Universal Robots PolyScope program: pos5.urp

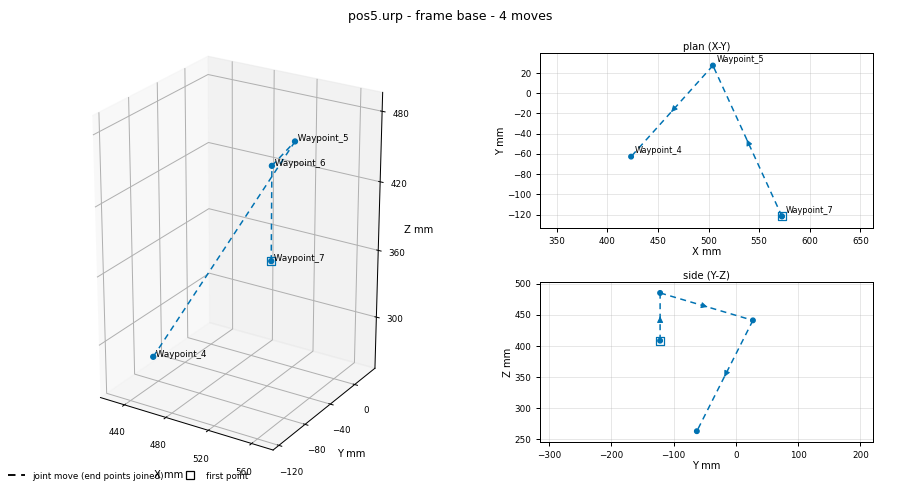
[picture p0: tool path of pos5.urp in frame base, 4 of 4 moves have a stored position in this frame; points joined in program order, loops and branches not executed]
Program pos5 (installation=default directory=/programs/Nicolas_Arteaga/quality createdIn=5.12.4.1101661 lastSavedIn=5.12.4.1101661 robotSerialNumber=20225502378)
Calibrated DH parameters: a=[0.00022, -0.425328, -0.389701, 0.000059, 0.000065, 0]; d=[0.162608, 0.803456, 9.992211, -10.662202, 0.099702, 0.099559]; alpha=[1.570756, 0.001543, 0.004316, 1.570651, -1.570122, 0]; deltaTheta=[0, 0.002917, 0.116094, -0.119008, 0, -0.000001]
Robot Program (runOnlyOnce=true)
  MoveJ speed 60 deg/s, acceleration 80 deg/s^2 (useActiveTCP=true) feature=Base
    Waypoint Waypoint_7: TCP in base x=572.475 y=-121.659 z=408.694 mm, rx=-1.467 ry=0.8075 rz=-0.784 rad; joints [121.622, -70.655, 92.719, 71.319, 2.368, 86.104] deg; TCP offset x=0 y=0 z=191.5 mm, rx=0 ry=0 rz=0 rad
    Waypoint Waypoint_6: TCP in base x=572.488 y=-121.624 z=485.395 mm, rx=-1.4669 ry=0.8076 rz=-0.7838 rad; joints [121.615, -73.605, 85.33, 82.996, 2.356, 84.774] deg; TCP offset x=0 y=0 z=191.5 mm, rx=0 ry=0 rz=0 rad
    Waypoint Waypoint_5: TCP in base x=504.298 y=27.412 z=441.351 mm, rx=-2.1458 ry=0.2085 rz=-0.4478 rad; joints [135.899, -74.63, 77.655, 112.181, 35.14, 43.687] deg; TCP offset x=0 y=0 z=191.5 mm, rx=0 ry=0 rz=0 rad
    Waypoint Waypoint_4: TCP in base x=423.421 y=-62.632 z=263.327 mm, rx=-2.7082 ry=-1.5112 rz=-0.0977 rad; joints [150.411, -75.414, 78.345, 87.06, 85.5, 2.039] deg
    'measure pressure pos1'
